# EPICS substitutions: modules/event/evrSupport/Db/ioc/IOC-IN20-LS17evr.substitutions
#==============================================================================
#
# Abs:  LCLS EVR IOC records for IN20 LS17
#
# Name: IOC-IN20-LS17evr.substitutions
#
#==============================================================================
#
file evrLSXX.db
{
pattern { DEVICE        }
	{ EVR:IN20:LS17 }
}
